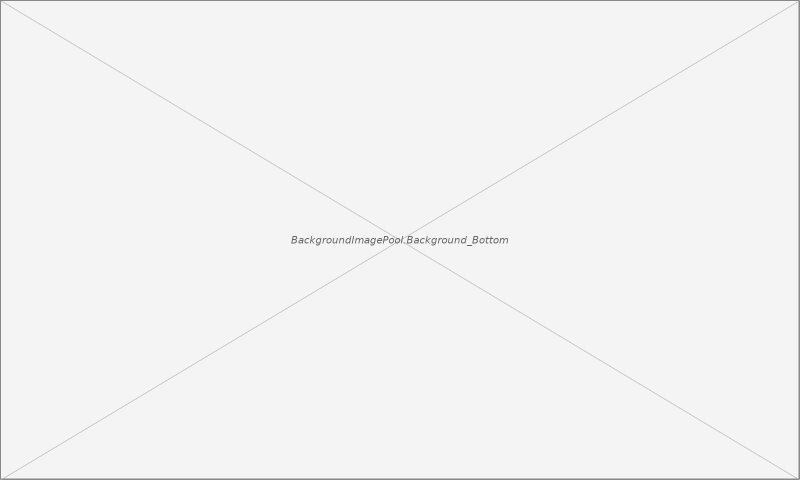
VISUALIZATION BackgroundNoButton  // 800x480
    Image (0,0 800x480), invisible if: SystemBase.bSystemOK, input disabled if: SystemBase.bSystemOK, image: BackgroundImagePool.Emergency Stop Active
    Image (0,0 800x480), image: BackgroundImagePool.Background_Bottom
END_VISUALIZATION

(* stored: Version 1.1.0.1, ProductVersion 3.1.4024.5
   Visu BackgroundNoButton: Id {7b934ca9-86fe-4224-81d7-f07b866cae24} *)
